INTERFACE I_RecipeBuilder

METHOD Build : BOOL
VAR_INPUT
    PanelWidth           : REAL;
    PanelLength          : REAL;
    PanelHeight          : REAL;
    CuttingOverpass      : REAL;
    RailHeightCorrection : REAL;
END_VAR
VAR_OUTPUT
    // Zwracamy wyliczone segmenty i ich ilość
    SegmentsGroove       : ARRAY[1..32] OF ST_CutSegment;
    SegmentsToGroove     : INT;
    
    SegmentsCutX         : ARRAY[1..32] OF ST_CutSegment;
    SegmentsToCutX       : INT;
    
    SegmentsCutY         : ARRAY[1..32] OF ST_CutSegment;
    SegmentsToCutY       : INT;
END_VAR
END_METHOD

END_INTERFACE

(* stored: Version 1.1.0.1, ProductVersion 3.1.4024.15
   Itf I_RecipeBuilder: Id {36800402-6cf0-4647-81a8-eb2cedcd2dc1}
   Method Build: Id {c09be119-3937-4a1a-9b08-f0b7fdecc5a6} *)
